(* CODESYS project ST1.project

Project tree, tasks and I/O mapping:
  Device : CODESYS Control Win V3, 3S - Smart Software Solutions GmbH, order no. 305021, version 3.5.10.30
    application Application
      libraries: Standard, * (System)
      task MainTask (cyclic, interval t#20ms, priority 1) calls PLC_PRG
      task VISU_TASK (cyclic, interval 100 ms, priority 31) calls VisuElems.Visu_Prg
      program PLC_PRG [ST]
      visualisation Visualization
  text list GlobalTextList
*)

// Device/Application/PLC_PRG
PROGRAM PLC_PRG
VAR
	Contact1: BOOL;
	Coil1: BOOL;
END_VAR

// This is a comment
(* This is another comment *)
IF Contact1 = TRUE THEN;
	Coil1 := TRUE;
ELSE;
	Coil1 := FALSE;
END_IF;

END_PROGRAM

// Device/Application/Visualization
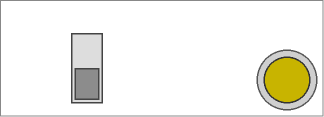
VISUALIZATION Visualization  // 324x117
    Lamp1 (252,45 70x70), variable: PLC_PRG.Coil1, style: Lamp-Lamp1-Yellow
    DipSwitch (52,33 70x70), variable: PLC_PRG.Contact1, behaviour: TOGGLE, style: Switch-DipSwitch-Gray
END_VISUALIZATION
